// TwinCAT 3 PLC project Slider
// ProgramVersion: 3.1.4024.0
// libraries:
//   Tc2_MC2, * (Beckhoff Automation GmbH)
//   Tc2_Standard, * (Beckhoff Automation GmbH)
//   Tc2_System, * (Beckhoff Automation GmbH)
//   Tc3_Module, * (Beckhoff Automation GmbH)
// project tree:
//   DUTs/Cell/ ST_CELL.TcDUT, E_CMD_CELL.TcDUT
//   DUTs/CM/ E_CM_SERVO_CMD.TcDUT, ST_CM_SERVO.TcDUT, ST_CM_SERVO_CMD.TcDUT, ST_CM_SERVO_STS.TcDUT
//   DUTs/CM/Servo/ fbCmServo.TcPOU
//   DUTs/EM/ E_CMD.TcDUT, E_Function.TcDUT, E_Status.TcDUT, ST_CONFIG.TcDUT, ST_DATA.TcDUT, ST_EM.TcDUT, ST_MACHINE.TcDUT
//   DUTs/UN/ ST_UN.TcDUT
//   DUTs/UTIL/ E_DIRECTION.TcDUT, E_pos.TcDUT, STATUS_HMI.TcDUT
//   / GlobalTextList.TcGTLO, PlcTask.TcTTO, Visualization Manager.TcVMO (not stored)
//   GVLs/ Counters.TcGVL, GVL.TcGVL
//   POUs/ MAIN.TcPOU
//   POUs/Module/ fbEM.TcPOU, fbSliderEM.TcPOU, fbSliderWithGripperEM.TcPOU, fbXYMoverEM.TcPOU
//   POUs/Sim/ fbSignalSimPiotr.TcPOU, fbSignalSimSlider.TcPOU, fbSignalSimSliderWithGripper.TcPOU, fbSignalSimXYMover.TcPOU
//   POUs/UN/ fbTaskPatrykUN.TcPOU, fbTaskPiotrUN.TcPOU, fbUN.TcPOU
//   VISUs/ VisuPiotrUN.TcVIS
// real-time tasks:
//   TASK PlcTask: cycle T#10ms, priority 20, ADS port 350
// motion (NC):
//   TASK NC-Task 1 SAF: cycle T#2ms, priority 4, ADS port 501
//   TASK NC-Task 1 SVB: cycle T#10ms, priority 8, ADS port 511
//   AXIS Axis 1 (id 1)
//     OtherSettings: AllowMotionCmdToSlave=true
//     encoder EncType=1
//     drive DrvType=5
//       Analog: TorqueSetpointScale=10, ScaleFactorActTorque=0.1
//       TimeComp: TaskDelayCycles=1
//     controller CtrType=1
//       CtrPara: PriorControlFactor=1
//         Observer: BandWidth=20

CONFIGURATION Slider
    RESOURCE PLC ON TwinCAT3
        TASK PlcTask(INTERVAL := T#10ms, PRIORITY := 20);
        PROGRAM MAIN WITH PlcTask : MAIN;
    END_RESOURCE
END_CONFIGURATION

// ---- DUTs/Cell/ST_CELL.TcDUT
TYPE ST_CELL :
STRUCT
	Cmd : E_CMD_CELL;
	PlaceObject : ARRAY[1..5] OF BOOL; 
END_STRUCT
END_TYPE

// ---- DUTs/Cell/E_CMD_CELL.TcDUT
{attribute 'qualified_only'}
{attribute 'strict'}
TYPE E_CMD_CELL :
(
	STOP := 0,
	START,
	ABORT
);
END_TYPE

// ---- DUTs/CM/E_CM_SERVO_CMD.TcDUT
{attribute 'qualified_only'}
{attribute 'strict'}
TYPE E_CM_SERVO_CMD :
(
	idle := 0,
	reset,
	powerDisable,
	powerEnable,
	brakeDisable,
	brakeEnable,
	halt,
	moveVel,
	moveRel,
	moveAbs,
	moveMod,
	moveHome,
	jogP,
	jogN,
	jogStop
);
END_TYPE

// ---- DUTs/CM/ST_CM_SERVO.TcDUT
TYPE ST_CM_SERVO :
STRUCT
	cmd: ST_CM_SERVO_CMD;
	sts: ST_CM_SERVO_STS;
END_STRUCT
END_TYPE

// ---- DUTs/CM/ST_CM_SERVO_CMD.TcDUT
TYPE ST_CM_SERVO_CMD :
STRUCT
	cmd : E_CM_SERVO_CMD;
	start : BOOL;
END_STRUCT
END_TYPE

// ---- DUTs/CM/ST_CM_SERVO_STS.TcDUT
TYPE ST_CM_SERVO_STS :
STRUCT
	done: BOOL;
	outPos: BOOL;
	nearPos: BOOL;
	homed: BOOL;
	power: BOOL;
	error: BOOL;
	errorCode: UDINT;
	pos: REAL;
END_STRUCT
END_TYPE

// ---- DUTs/EM/E_CMD.TcDUT
// Enumerator containing em commands
{attribute 'qualified_only'}
{attribute 'strict'}
TYPE E_CMD :
(
	reset:=1,
	start,
	stop,
	hold,
	unhold,
	suspend,
	unsuspend,
	abort,
	clear,
	powerOn
);
END_TYPE

// ---- DUTs/EM/E_Function.TcDUT
// Enumerator containing general function of module
{attribute 'qualified_only'}
{attribute 'strict'}
{attribute 'to_string'}
TYPE E_Function :
(
	None,
	eSlider,
	eSliderWithGripper,
	eXYMover
);
END_TYPE

// ---- DUTs/EM/E_Status.TcDUT
// Enumerator contains packml state, unfortunatly named status
{attribute 'qualified_only'}
{attribute 'strict'}
TYPE E_Status :
(
	undefined:=0,
	clearing,
	stopped,
	starting,
	idle,
	suspended,
	execute,
	stopping,
	aborting,
	aborted,
	holding,
	held,
	unholding,
	suspending,
	unsuspending,
	resetting,
	completing,
	completed
);
END_TYPE

// ---- DUTs/EM/ST_CONFIG.TcDUT
// Structure config
{attribute 'qualified_only'}
{attribute 'strict'}
TYPE ST_CONFIG :
STRUCT
	Functionality : E_Function;
	Data : ST_DATA;
END_STRUCT
END_TYPE

// ---- DUTs/EM/ST_DATA.TcDUT
// Structure data contains inputs/outputs/axies
TYPE ST_DATA :
STRUCT
	I : REFERENCE TO ARRAY[1..10] OF BOOL;
	Q : REFERENCE TO ARRAY[1..10] OF BOOL;
	Axis : ARRAY[1..10] OF AXIS_REF;
	pick_pos :INT ; 					// Q CMD from where girpper picks
	drop_pos: INT ;						// Q CMD to where gripper moves for drop
	act_pos: INT;						// I actual position from of gripper
	give_pos: INT;						// writes value to servo_handle // simulator 
	takeObject : BOOL;
	objectSensor : BOOL;
END_STRUCT
END_TYPE

// ---- DUTs/EM/ST_EM.TcDUT
// Base structure em
TYPE ST_EM :
STRUCT
	Config : ST_CONFIG;
	Cmd : E_CMD;
	Status : E_Status;
	SequenceStep: INT;
	StatusHMI : STATUS_HMI;
END_STRUCT
END_TYPE

// ---- DUTs/EM/ST_MACHINE.TcDUT
// Utility structure to reference to fbEM
TYPE ST_MACHINE :
STRUCT
	fbEM : REFERENCE TO fbEM;
END_STRUCT
END_TYPE

// ---- DUTs/UN/ST_UN.TcDUT
// For now empty structure to build master for em-s
TYPE ST_UN :
STRUCT
	Cmd : E_CMD;
	Status : E_Status;
END_STRUCT
END_TYPE

// ---- DUTs/UTIL/E_DIRECTION.TcDUT
{attribute 'qualified_only'}
{attribute 'strict'}
TYPE E_DIRECTION :
(
	Left,
	Right,
	Up,
	Down,
	Downstream,
	Upstream
);
END_TYPE

// ---- DUTs/UTIL/E_pos.TcDUT
{attribute 'qualified_only'}
{attribute 'strict'}
TYPE E_pos :
(
	base := 0,
	one,
	two,
	three,
	four
	
);
END_TYPE

// ---- DUTs/UTIL/STATUS_HMI.TcDUT
TYPE STATUS_HMI :
STRUCT
	isMoving : BOOL;
	movingToPosition : INT;
	currentPosition : INT;
	movingDirection : E_DIRECTION;
	hasObject : BOOL;
	alarm : BOOL;
	alarmText : STRING;
	undefined : BOOL;
END_STRUCT
END_TYPE

// ---- GVLs/Counters.TcGVL
{attribute 'qualified_only'}
VAR_GLOBAL CONSTANT
	SliderEMNo : INT := 1;
	SliderWithGripperEMNo : INT := 1;
	XYMoverEMNo : INT := 2;
	
	packmlUnLast : INT := 1;
	packmlEmLast : INT := SliderEMNo + SliderWithGripperEMNo + XYMoverEMNo;
END_VAR

// ---- GVLs/GVL.TcGVL
// Global list with inputs/outputs to control and force variables
{attribute 'qualified_only'}
VAR_GLOBAL
	axis : AXIS_REF;
	aInput : ARRAY[1..10] OF ARRAY[1..10] OF BOOL;
	aOutput : ARRAY[1..10] OF ARRAY[1..10] OF BOOL;
	
	Input : ARRAY[1..10] OF BOOL;
	Output : ARRAY[1..10] OF BOOL;
END_VAR

// ---- POUs/MAIN.TcPOU
PROGRAM MAIN
VAR
	un : ST_UN;
	cell : ST_CELL;
	fbTaskPiotrUN : fbTaskPiotrUN;
	
	fb : fbSliderEM;
	em : ST_EM;
	
	START : BOOL;
	STOP : BOOL;
	ABORT : BOOL;
END_VAR

//cell.Cmd := E_CMD_CELL.START; 	// Selected as constant START to work in loop
//cell.PlaceObject := TRUE;		// Selected as constant placing object at input to work in loop

IF START THEN
	cell.Cmd := E_CMD_CELL.START;
	START := FALSE;
ELSIF STOP THEN
	cell.Cmd := E_CMD_CELL.STOP;
	STOP := FALSE;
ELSIF ABORT THEN
	cell.Cmd := E_CMD_CELL.ABORT;
	ABORT := FALSE;
END_IF

fbTaskPiotrUN(un := un, cell := cell, EnableSim := TRUE);

END_PROGRAM

// ---- POUs/UN/fbTaskPiotrUN.TcPOU
FUNCTION_BLOCK fbTaskPiotrUN EXTENDS fbUN
VAR
	// Arrays with 'em' universal structure and 'fbEM' containing ST_MACHINE structure which contains of references to fbEM function block
	em : ARRAY[1..Counters.packmlEmLast] OF ST_EM;
	fbEM : ARRAY[1..Counters.packmlEmLast] OF ST_MACHINE;
	
	// Array containing all instances fo fbSliderEM with its own iterator
	SliderEM : ARRAY[1..Counters.SliderEMNo] OF fbSliderEM;
	iSliderEM : DINT := 1;
	
	// Array containing all instances fo fbSliderWithGripperEM with its own iterator
	SliderWithGripperEM : ARRAY[1..Counters.SliderWithGripperEMNo] OF fbSliderWithGripperEM;
	iSliderWithGripperEM : DINT := 1;
	
	// Array containing all instances fo fbXYMoverEM with its own iterator
	XYMoverEM : ARRAY[1..Counters.XYMoverEMNo] OF fbXYMoverEM;
	iXYMoverEM : DINT := 1;
	
	fbSignalSimPiotr : fbSignalSimPiotr;
	
	i : DINT;
	j : DINT;
	State : INT := 0;
	StoppedState : INT := 0;
	declareIterator : DINT;
	moduleWorkIterator : DINT;
	initialConfig: BOOL := TRUE;
	svTime : TIME := T#15S;
	oTime : TIME := T#1S;
	supervisionTimer: TON;
	objectTimer: TON;
	objectWhichStopped : DINT := 0;
	takeObjectCounter : USINT;
	stoppedBy : STRING := '';
	stoppedByTemp : STRING;
	oneAlarm: BOOL;
END_VAR

// fbEM and em array number:
// 1 <- XYMovers
// 2 <- SliderWithGripper
// 3 <- XYMover
// 4 <- Slider
// 5 <- Slider

////////////////////////////////////////////////////////////////////////////////////////////////////////////////////////////
// All init configuration done here
IF initialConfig THEN
	initialConfig := FALSE;
	// Specifing module type of each module in array
	em[1].Config.Functionality := E_Function.eXYMover;
	em[2].Config.Functionality := E_Function.eSliderWithGripper;
	em[3].Config.Functionality := E_Function.eXYMover;
	em[4].Config.Functionality := E_Function.eSlider;
	em[5].Config.Functionality := E_Function.eSlider;

	// FOR loop to specify config for each module
	FOR declareIterator := 1 TO Counters.packmlEmLast DO
		em[declareIterator].Config.Data.I REF= GVL.aInput[declareIterator];
		em[declareIterator].Config.Data.Q REF= GVL.aOutput[declareIterator];

		CASE em[declareIterator].Config.Functionality OF
			E_Function.eSlider:
				fbEM[declareIterator].fbEM REF= SliderEM[iSliderEM];
				iSliderEM := iSliderEM + 1;
			E_Function.eSliderWithGripper:
				fbEM[declareIterator].fbEM REF= SliderWithGripperEM[iSliderWithGripperEM];
				iSliderWithGripperEM := iSliderWithGripperEM + 1;
			E_Function.eXYMover:
				fbEM[declareIterator].fbEM REF= XYMoverEM[iXYMoverEM];
				iXYMoverEM := iXYMoverEM + 1;
		END_CASE
	END_FOR
	
	em[2].Config.Data.pick_pos := 3;
	em[2].Config.Data.drop_pos := 2;
	
	supervisionTimer.PT := svTime;
	objectTimer.PT := oTime;
END_IF

////////////////////////////////////////////////////////////////////////////////////////////////////////////////////////////
// Modules work loop (idk yet if is better to have it at the beggining or bottom of UN)
FOR moduleWorkIterator := 1 TO Counters.packmlEmLast DO
	fbEM[moduleWorkIterator].fbEM(em := em[moduleWorkIterator], un := un, EnableSim := EnableSim, CmdSim := FALSE);
END_FOR

////////////////////////////////////////////////////////////////////////////////////////////////////////////////////////////

fbSignalSimPiotr(em := em, State := State, EnableSim := EnableSim);

IF supervisionTimer.Q THEN
	stoppedBy := 'Supervision';
	supervisionTimer(IN := FALSE);
	cell.Cmd := E_CMD_CELL.STOP;
END_IF

FOR j := 1 TO Counters.packmlEmLast DO
	IF NOT em[j].Config.Data.takeObject AND em[j].Config.Data.objectSensor THEN
		objectTimer(IN := TRUE);
		objectWhichStopped := j;
	ELSIF objectWhichStopped = j
	AND ((em[j].Config.Data.takeObject AND em[j].Config.Data.objectSensor)
	OR (NOT em[j].Config.Data.takeObject AND NOT em[j].Config.Data.objectSensor)) THEN
		objectWhichStopped := 0;
		objectTimer(IN := FALSE);
		oneAlarm := FALSE;
	END_IF
END_FOR

IF objectTimer.Q THEN
	cell.Cmd := E_CMD_CELL.STOP;
	IF NOT oneAlarm THEN
		stoppedBy := CONCAT('Object at em: ', DINT_TO_STRING(ObjectWhichStopped));
		oneAlarm := TRUE;
	END_IF
END_IF

IF cell.Cmd = E_CMD_CELL.STOP AND State < 2000 THEN
	StoppedState := State;
	State := 2000;
END_IF

IF cell.Cmd = E_CMD_CELL.ABORT AND State < 1000 THEN
	stoppedBy := 'ABORT Button';
	StoppedState := 0;
	State := 1000;
END_IF

CASE State OF
	0:	un.Status := E_Status.undefined;
		em[2].Config.Data.pick_pos := 3;
		em[2].Config.Data.drop_pos := 2;
		State := 5;
	
	5:	// Waiting for every EM to become idle state
		FOR i := 1 TO Counters.packmlEmLast DO
			IF NOT (em[i].Status = E_Status.idle) THEN
				un.Cmd := E_CMD.reset;
				RETURN;
			END_IF
		END_FOR
		un.Status := E_Status.idle;
		State := 10;
	
	10:	IF cell.Cmd = E_CMD_CELL.START THEN
			stoppedBy := '';
			un.Cmd := E_CMD.start;
			un.Status := E_Status.starting;
			State := 20;
		END_IF
	
	20:	// Waiting for every EM to be in execute or starting state
		FOR i := 1 TO Counters.packmlEmLast DO
			IF NOT (em[i].Status = E_Status.execute OR em[i].Status = E_Status.starting) THEN
				RETURN;
			END_IF
		END_FOR
		State := 30;
		
	30:	// Start of my specific task (all modules stays in execute)
		// input -> XY1 -> SWG -> XY2 -> S1 -> SWG -> S2 -> output
		IF (em[1].SequenceStep = 20		// XY1
		AND cell.PlaceObject)			// Object input signal
		THEN
			cell.PlaceObject := FALSE;
			em[1].Config.Data.takeObject := TRUE;
			State := 40;
		END_IF
		
		IF StoppedState <> 0 AND StoppedState < 1000 THEN
			State := StoppedState;
			StoppedState := 0;
		END_IF
		
	40:	// XY1 -> SWG -> XY2 -> S1 -> SWG -> S2 -> output
		supervisionTimer(IN := TRUE);
		
		IF em[1].SequenceStep = 60		// XY1
		AND em[2].SequenceStep = 40		// SWG
		THEN
			em[1].Config.Data.takeObject := FALSE;
			em[2].Config.Data.takeObject := TRUE;
			
			State := 50;
			supervisionTimer(IN := FALSE);
		END_IF
		
	50: // SWG -> XY2 -> S1 -> SWG -> S2 -> output
		supervisionTimer(IN := TRUE);
		
		IF em[2].SequenceStep = 43		// SWG
		AND em[3].SequenceStep = 20		// XY2
		THEN
			em[2].Config.Data.takeObject := FALSE;
			em[3].Config.Data.takeObject := TRUE;
			
			em[2].Config.Data.pick_pos := 4;
			State := 60;
			supervisionTimer(IN := FALSE);
		END_IF
		
	60: // XY2 -> S1 -> SWG -> S2 -> output
		supervisionTimer(IN := TRUE);
		
		IF em[3].SequenceStep = 60		// XY2
		AND em[4].SequenceStep = 50		// S1
		THEN
			em[3].Config.Data.takeObject := FALSE;
			em[4].Config.Data.takeObject := TRUE;
			
			em[2].Config.Data.drop_pos := 1;
			State := 70;
			supervisionTimer(IN := FALSE);
		END_IF
		
	70:	// S1 -> SWG -> S2 -> output
		supervisionTimer(IN := TRUE);
		
		IF em[2].SequenceStep = 40		// SWG
		AND em[4].SequenceStep = 70		// S1
		THEN
			em[4].Config.Data.takeObject := FALSE;
			em[2].Config.Data.takeObject := TRUE;
			
			State := 80;
			supervisionTimer(IN := FALSE);
		END_IF
		
	80:	// SWG -> S2 -> output
		supervisionTimer(IN := TRUE);
		
		IF em[2].SequenceStep = 43		// SWG
		AND em[5].SequenceStep = 50		// S2
		THEN
			em[2].Config.Data.takeObject := FALSE;
			em[5].Config.Data.takeObject := TRUE;
			
			em[2].Config.Data.pick_pos := 3;
			State := 90;
			supervisionTimer(IN := FALSE);
		END_IF
		
	90:	// S2 -> output
		supervisionTimer(IN := TRUE);
		IF em[5].SequenceStep = 70 THEN
			em[2].Config.Data.drop_pos := 2;
			State := 100;
			supervisionTimer(IN := FALSE);
		END_IF
		
	100: // output
		IF NOT em[5].Config.Data.objectSensor THEN
			em[5].Config.Data.takeObject := FALSE;
			State := 30;
		END_IF
		
	1000:
		un.Cmd := E_CMD.abort;
		un.Status := E_Status.aborting;
		FOR i := 1 TO Counters.packmlEmLast DO
			IF NOT (em[i].Status = E_Status.aborted) THEN
				RETURN;
			END_IF
		END_FOR
		State := 1010;
	
	1010:
		IF cell.Cmd = E_CMD_CELL.START THEN
			un.Cmd := E_CMD.clear;
			State := 2000;
		END_IF

	2000:
		un.Cmd := E_CMD.stop;
		un.Status := E_Status.stopping;
		supervisionTimer(IN := FALSE);
		objectTimer(IN := FALSE);
		FOR i := 1 TO Counters.packmlEmLast DO
			IF em[i].Status <> E_Status.stopped THEN
				RETURN;
			END_IF
		END_FOR
		un.Status := E_Status.stopped;
		State := 2010;
	
	2010:
		IF cell.Cmd = E_CMD_CELL.START THEN
			State := 5;
		END_IF	
END_CASE

// Do not write anything here, it will not execute everytime due to RETURN command used in case

END_FUNCTION_BLOCK

// ---- POUs/UN/fbUN.TcPOU
FUNCTION_BLOCK fbUN
VAR_IN_OUT
	un : ST_UN;
	cell : ST_CELL;
END_VAR
VAR_INPUT
	EnableSim : BOOL;
END_VAR

END_FUNCTION_BLOCK

// ---- POUs/Module/fbEM.TcPOU
FUNCTION_BLOCK fbEM
VAR_IN_OUT
	em : ST_EM;
	un : ST_UN;
END_VAR

VAR_INPUT
	EnableSim : BOOL;
	CmdSim : BOOL := TRUE;
END_VAR

VAR
	emCmdOld: E_CMD;
END_VAR

// Empty for now universal basic em class, every module needs to extends this to ensure compatibility

ACTION GetUnCmd:
IF emCmdOld <> un.Cmd THEN
	emCmdOld := un.Cmd;
	em.Cmd := un.Cmd;
END_IF
END_ACTION

END_FUNCTION_BLOCK

// ---- POUs/Module/fbSliderEM.TcPOU
FUNCTION_BLOCK fbSliderEM EXTENDS fbEM
VAR_INPUT
	UnknownStartPosition : BOOL := FALSE;
	StartOnOtherSide : BOOL := FALSE;
END_VAR

VAR
	bSliderSide : BOOL;
	XYMoverActualStep: INT;
	fbSignalSim : fbSignalSimSlider;
	timer : TON;
	timerPT : TIME := T#2S;
END_VAR

VAR RETAIN
	State : INT := 0;
END_VAR

(*
	Input/Output mapping
	I[1] <- Siłownik pozycja 1 (wsunięty) 
	I[2] <- Siłownik pozycja 2 (wysunięty)
	I[3] <- Czujnik obecności obiektu (na pozycji 1 (wsunięty)) 
	Q[1] <- Wysuń siłownik (do pozycji 2)
	Q[2] <- Wsuń siłownik (do pozycji 1)
*)

GetUnCmd();
fbSignalSim(
	em := em,
	EnableSim := EnableSim,
	UnknownStartPosition := UnknownStartPosition,
	StartOnOtherSide := StartOnOtherSide,
	CmdSim := CmdSim
);
timer(PT := timerPT);

IF em.Config.Functionality = E_Function.eSlider THEN
	IF State >= 15 AND em.Cmd = E_CMD.abort THEN
		State := 5;
	END_IF
	
	IF State >= 35 AND em.Cmd = E_CMD.stop THEN
		State := 15;
	END_IF

	CASE State OF
		0:	em.StatusHMI.isMoving := FALSE;
			em.StatusHMI.undefined := TRUE;
			IF em.Config.Data.I[1] OR em.Config.Data.I[2] THEN
				State := 1;
				em.StatusHMI.undefined := FALSE;
			ELSE
				em.Status := E_Status.undefined;
				State := 20;
			END_IF
			
		1:	IF em.Config.Data.I[2] THEN
				bSliderSide := TRUE;
				em.StatusHMI.currentPosition := 2;
			ELSE
				em.StatusHMI.currentPosition := 1;
			END_IF
			State := 40;
		
		5:	em.Status := E_Status.aborting;
			em.Config.Data.Q[1] := FALSE;
			em.Config.Data.Q[2] := FALSE;
			em.StatusHMI.isMoving := FALSE;
			em.StatusHMI.undefined := TRUE;
			State := 7;
			
		7:	em.Status := E_Status.aborted;
			State := 10;
			
		10:	IF em.Cmd = E_CMD.clear THEN
				em.Status := E_Status.clearing;
				em.StatusHMI.undefined := FALSE;
				State := 20;
			END_IF
			
		15: em.Status := E_Status.stopping;
			em.Config.Data.Q[1] := FALSE;
			em.Config.Data.Q[2] := FALSE;
			em.StatusHMI.isMoving := FALSE;
			em.StatusHMI.undefined := FALSE;
			State := 20;
			
		20:	em.Status := E_Status.stopped;
			State := 30;
			
		30:	IF em.Cmd = E_CMD.reset THEN
				em.Status := E_Status.resetting;
				em.Config.Data.Q[1] := FALSE;
				em.Config.Data.Q[2] := TRUE;
				em.StatusHMI.isMoving := TRUE;
				em.StatusHMI.movingDirection := E_DIRECTION.Upstream;
				em.StatusHMI.movingToPosition := 1;
				State := 35;
			END_IF
			
		35:	IF em.Config.Data.I[1] THEN
				em.StatusHMI.isMoving := FALSE;
				em.Config.Data.Q[2] := FALSE;
				bSliderSide := FALSE;
				State := 40;
			END_IF
			
		40:	em.Status := E_Status.idle;
			IF em.Cmd = E_CMD.start THEN
				State := 45;
			END_IF
			
		45:	em.Status := E_Status.Starting;
			State := 50;
			
			// Execute direction
		50:	em.Status := E_Status.execute;
			IF bSliderSide AND NOT em.Config.Data.I[3] THEN
				timer(IN := TRUE);
				State := 52;
			ELSIF em.Config.Data.I[3] THEN
				timer(IN := TRUE);
				State := 55;
			END_IF
			
		52: IF timer.Q THEN
				em.StatusHMI.movingDirection := E_DIRECTION.Upstream;
				em.StatusHMI.movingToPosition := 1;
				em.StatusHMI.undefined := FALSE;
				timer(IN := FALSE);
				em.Config.Data.Q[2] := TRUE;
				State := 60;
			END_IF	
			
		55: IF timer.Q THEN
				em.StatusHMI.movingDirection := E_DIRECTION.Downstream;
				em.StatusHMI.movingToPosition := 2;
				em.StatusHMI.undefined := FALSE;
				timer(IN := FALSE);
				em.Config.Data.Q[1] := TRUE;
				State := 60;
			END_IF	
			
			// Main execute
		60:	IF em.Cmd = E_CMD.hold THEN
				em.StatusHMI.undefined := TRUE;
				em.Status := E_Status.holding;
				State := 200;
			ELSIF em.Cmd = E_CMD.suspend THEN
				em.StatusHMI.undefined := TRUE;
				em.Status := E_Status.suspending;
				State := 300;
			END_IF
			
			IF em.Config.Data.Q[2] AND em.Config.Data.I[1] THEN
				em.Config.Data.Q[2] := FALSE;
				bSliderSide := FALSE;
				State := 50;
			END_IF
			
			IF em.Config.Data.Q[1] AND em.Config.Data.I[2] THEN
				bSliderSide := TRUE;
				State := 70;
			END_IF
			
		70:	IF NOT em.Config.Data.I[3] THEN
				em.Config.Data.Q[1] := FALSE;
				State := 50;
			END_IF
			
		200:em.Status := E_Status.held;
			em.Config.Data.Q[1] := FALSE;
			em.Config.Data.Q[2] := FALSE;
			em.StatusHMI.undefined := TRUE;
			IF em.Cmd = E_CMD.unhold THEN
				em.Status := E_Status.unholding;
				State := 50;
			END_IF
			
		300:em.Status := E_Status.suspended;
			em.Config.Data.Q[1] := FALSE;
			em.Config.Data.Q[2] := FALSE;
			em.StatusHMI.undefined := TRUE;
			IF em.Cmd = E_CMD.unsuspend THEN
				em.Status := E_Status.unsuspending;
				State := 50;
			END_IF
	END_CASE
END_IF

em.SequenceStep := State;
em.Config.Data.objectSensor REF= em.Config.Data.I[3];

IF em.Config.Data.Q[1] XOR em.Config.Data.Q[2] THEN
	em.StatusHMI.isMoving := TRUE;
ELSIF em.Config.Data.Q[1] AND em.Config.Data.Q[2] THEN
	em.StatusHmi.isMoving := FALSE;
	em.StatusHMI.undefined := TRUE;
	em.StatusHMI.alarm := TRUE;
	em.StatusHMI.alarmText := 'Both actuators are operating';
ELSE
	em.StatusHmi.isMoving := FALSE;
	em.StatusHMI.undefined := FALSE;
	em.StatusHMI.alarm := FALSE;
	em.StatusHMI.alarmText := '';
END_IF

IF em.Config.Data.I[3] THEN
	em.StatusHMI.hasObject := TRUE;
ELSE
	em.StatusHMI.hasObject := FALSE;
END_IF

IF em.Config.Data.I[1] THEN
	em.StatusHMI.currentPosition := 1;
ELSIF em.Config.Data.I[2] THEN
	em.StatusHMI.currentPosition := 2;
ELSE
	em.StatusHMI.currentPosition := 0;
END_IF

END_FUNCTION_BLOCK

// ---- POUs/Sim/fbSignalSimSlider.TcPOU
FUNCTION_BLOCK fbSignalSimSlider
VAR_IN_OUT
	em : ST_EM;
END_VAR
VAR_INPUT
	EnableSim : BOOL;
	UnknownStartPosition : BOOL := FALSE;
	StartOnOtherSide : BOOL := FALSE;
	CmdSim : BOOL := true;
END_VAR
VAR
	InitialConfig : BOOL := TRUE;
	timers : ARRAY[1..10] OF TON;
	duration : TIME := T#5S;
	elapsed : TIME;
	OtherSide : BOOL := FALSE;
END_VAR

IF EnableSim THEN
	IF InitialConfig THEN
		InitialConfig := FALSE;
		IF NOT UnknownStartPosition THEN
			IF StartOnOtherSide THEN
				em.Config.Data.I[2] := TRUE;
				OtherSide := TRUE;
			ELSE
				em.Config.Data.I[1] := TRUE;
			END_IF
		ELSE
			em.Config.Data.I[1] := FALSE;
			em.Config.Data.I[2] := FALSE;
		END_IF
		
		timers[1].PT := timers[2].PT := timers[3].PT := timers[10].PT := duration;
		timers[4].PT := timers[5].PT := timers[6].PT := timers[7].PT := timers[8].PT := timers[9].PT := duration / 3;
	END_IF
	
	CASE em.SequenceStep OF
		10:	IF CmdSim THEN
				timers[5](in := TRUE);
			
				IF timers[5].Q THEN
					timers[5](in := FALSE);
					em.Cmd := E_CMD.clear;
				END_IF
			END_IF
	
		30:	IF CmdSim THEN
				timers[6](in := TRUE);
			
				IF timers[6].Q THEN
					timers[6](in := FALSE);
					em.Cmd := E_CMD.reset;	
				END_IF
			END_IF

		35:	timers[10](in := TRUE);
		
			IF timers[10].Q THEN
				timers[10](in := FALSE);
				em.Config.Data.I[1] := TRUE;
			END_IF
	
		40: IF CmdSim THEN
				timers[4](in := TRUE);
			
				IF timers[4].Q THEN
					timers[4](in := FALSE);
					em.Cmd := E_CMD.start;
				END_IF
			END_IF

		50:	IF CmdSim THEN
				IF NOT OtherSide AND em.Config.Data.I[1] THEN
					timers[1](in := TRUE); 
				END_IF
				
				IF timers[1].Q THEN
					timers[1](in := FALSE);
					em.Config.Data.I[3] := TRUE;
				END_IF
			END_IF
			
		60:	IF NOT OtherSide AND em.Config.Data.I[1] THEN
				timers[2](in := NOT timers[2].Q);
				em.Config.Data.I[1] := FALSE;
				em.Config.Data.I[2] := FALSE;
			ELSE
				timers[3](in := NOT timers[3].Q);
				em.Config.Data.I[1] := FALSE;
				em.Config.Data.I[2] := FALSE;
			END_IF
			
			IF timers[2].Q THEN
				timers[2](in := FALSE);
				em.Config.Data.I[2] := TRUE;
			END_IF
			
			IF timers[3].Q THEN
				timers[3](in := FALSE);
				em.Config.Data.I[1] := TRUE;
			END_IF
			
		70:	IF CmdSim THEN
				timers[1](in := TRUE);
				
				IF timers[1].Q THEN
					timers[1](in := FALSE);
					em.Config.Data.I[3] := FALSE;
				END_IF
			END_IF
			
		200:IF CmdSim THEN
				timers[8](in := TRUE);
			
				IF timers[8].Q THEN
					timers[8](in := FALSE);
					em.Cmd := E_CMD.unhold;	
				END_IF
			END_IF
		
		300:IF CmdSim THEN
				timers[9](in := TRUE);
			
				IF timers[9].Q THEN
					timers[9](in := FALSE);
					em.Cmd := E_CMD.unsuspend;	
				END_IF
			END_IF
	END_CASE

	OtherSide := FALSE;
END_IF

END_FUNCTION_BLOCK

// ---- POUs/Module/fbSliderWithGripperEM.TcPOU
FUNCTION_BLOCK fbSliderWithGripperEM EXTENDS fbEM
VAR
	i : INT;
	state : INT;
	initial: BOOL := TRUE;
	servo_GO: BOOL;
	
	fbSignalSim: fbSignalSimSliderWithGripper;
END_VAR
VAR_INPUT
	
END_VAR
VAR_OUTPUT
	
END_VAR

(*
THIS fb use IOs listed below
DATA.I[1] -> true when gripper closed
DATA.I[2] -> true when gripper opened
DATA.I[3] -> part present
DATA.Q[1] -> 1 CLOSE / 0 OPEN gripper
DATA.Q[3] -> SERVO_GO
DATA.pick_pos -> desired pick position
DATA.drop_pos -> desired drop position
DATA.act_pos -> actual postition ( resolved in SIM or SERVO_HANDLER)
DATA.give_pos -> moves desired position into SIM or SERVO_HANDLER)
*)

GetUnCmd();
fbSignalSim(
	em := em,
	EnableSim := EnableSim,
	CmdSim := CmdSim
);

IF initial THEN // AFTER START OF PLC ENTER Undefined state
	state:=0;
	//em.CMD := E_CMD.powerOn; //// MAKES SENSE? <- no it doesnt because you change input 
	initial:= FALSE;
	//	 em.Config.Data.pick_pos:=10; 
	//	 em.Config.Data.pick_pos:=200;
	
END_IF

IF em.CMD = E_CMD.abort THEN
	state:=65;
END_IF

IF em.CMD = E_CMD.stop THEN
	state:=70;
END_IF

CASE state OF
	
	0:		//RESETTING
		em.Status := E_Status.resetting;	
		
		
		IF  em.Config.Data.pick_pos = em.Config.Data.act_pos THEN   // ACTUAL POS READ FROM SERVO HANDLER / FOR NOW FROM SIGNAL SIM
				
				servo_GO:=FALSE;
				state :=30; // IF gripper at PICK_pos go to idle
		END_IF
		IF em.CMD = E_CMD.reset THEN 		
				em.Config.Data.give_pos:=em.Config.Data.pick_pos;
				servo_GO:=TRUE;
				
				//// IF gripper pos unknown move to PICK
				//SERVO_HANDLER HAS TO KNOW THE CASE STEP TO DECIDE WHERE TO MOVE 			 
				//HERE SIGNAL SIM HANDLE THIS		
		END_IF
		

	
	30:		//IDLE
		em.Status := E_Status.idle;
		IF em.CMD = E_CMD.start THEN 
			state :=40;
		END_IF
		

	40:		//EXECUTE.1
		em.Status := E_Status.execute;
				
		//Close gripper when part present
		IF em.Config.Data.I[3]  THEN 
			em.Config.Data.Q[1]:= TRUE; //CLOSE GRIPPER
		END_IF
		
		//When Gripper closed --> state 41
		IF em.Config.Data.I[1] = TRUE AND em.Config.Data.I[2]=FALSE THEN
			state:=41;
		END_IF

	41:		//EXECUTE.2 ORDER TO MOVE TO CHOOSEN POSITION
		em.Status := E_Status.execute;
		em.Config.Data.give_pos := em.Config.Data.drop_pos;
		servo_GO:=TRUE; 							
		IF em.Config.Data.act_pos = em.Config.Data.drop_pos THEN
		servo_GO:=FALSE;
		state:=42;										
		END_IF


	42:		//EXECUTE.3 OPEN GRIPPER
	
		em.Status := E_Status.execute;
		em.Config.Data.Q[1]:=FALSE; //OPEN GRIPPER
		IF em.Config.Data.I[1] = FALSE AND em.Config.Data.I[2]=TRUE THEN
			state:=43;
		END_IF
		
			
	43:		//EXECUTE.4 MOVING PICK_POS WITHOUT PART

		em.Status := E_Status.execute;
		IF NOT em.Config.Data.I[3]  
			AND em.Config.Data.act_pos =em.Config.Data.drop_pos THEN//when part gone
			em.Config.Data.give_pos:=em.Config.Data.pick_pos;
			servo_GO:=TRUE;//GO 
			//SERVO_HANDLER HAS TO KNOW THE CASE STEP TO DECIDE WHERE TO MOVE 			 
			//HERE SIGNAL SIM HANDLE THIS	
		END_IF
		
		IF em.Config.Data.act_pos = em.Config.Data.pick_pos THEN
			servo_GO:=FALSE;
			state:=40;
			//em.Config.Data.pick_pos:= -1;
			//em.Config.Data.drop_pos:= -1;
		END_IF
	
	
	65:		//ABORTED

		em.Status := E_Status.aborted;	
		servo_GO:=FALSE;
		IF em.CMD = E_CMD.clear THEN
			state := 70;
		END_IF;


	70: //STOPPED

		em.Status := E_Status.stopped;	
		servo_GO:=FALSE;
		IF em.CMD = E_CMD.reset THEN
			state:=0;
		END_IF

	
END_CASE



em.SequenceStep:=state;       //pass sequence step outside to SimSignal

em.Config.Data.Q[3]:=servo_GO;//Q[3] alias
em.Config.Data.objectSensor REF= em.Config.Data.I[3];




(*  SERVO HANDLER LOGIC
	IF SERVO_GO AND STATE = 0 THEN MOVE_TO_PICK_POS
	IF SERVO_GO AND STATE = 41 THEN MOVE_TO_DROP_POS
	IF SERVO_GO AND STATE = 44 THEN MOVE_TO_PICK_POS  *)

(*BEST MOMENT TO WRITE DESIRED pick_pos or drop_pos is STATE 30 or 40*)

END_FUNCTION_BLOCK

// ---- POUs/Sim/fbSignalSimSliderWithGripper.TcPOU
FUNCTION_BLOCK fbSignalSimSliderWithGripper
VAR_IN_OUT
	em : ST_EM; 
END_VAR
VAR_INPUT
	EnableSim : BOOL;
	CmdSim : BOOL := true;
END_VAR
VAR
	 
	i : int; 
	delay: ARRAY [1..10] OF TON;
END_VAR

delay[1](PT:=T#2S); delay[1].ET;//Open GRIPPER Movement Sim
delay[2](PT:=T#2S); delay[2].ET;//Close GRIPPER Movement SIm
delay[3](PT:=T#5S); delay[3].ET;// Moving  PICK_POS //DROP_POS
delay[4](PT:=T#4S); delay[4].ET;//CMD.Clear simulation
delay[5](PT:=T#4S); delay[5].ET;
delay[6](PT:=T#4S); delay[6].ET;
delay[7](PT:=T#4S); delay[7].ET;//OpenGRipp State 0
delay[9](PT:=T#2S); delay[9].ET;//CMD.clear
delay[10](PT:=T#2S);delay[10].ET;//CMD.reset

IF EnableSim THEN
		
	IF em.Cmd = E_CMD.abort THEN
		delay[9](IN:=TRUE);
	END_IF
	
	IF em.Cmd = E_CMD.stop THEN
		delay[10](IN:=TRUE);
	END_IF
	
	
	
	CASE em.SequenceStep OF
		
		0:		//Undefined state
				
			
				//Simulate CMD.clear button
			IF CmdSim THEN	
				IF delay[4].Q THEN
					delay[4](IN:=FALSE);
					em.Cmd:=E_CMD.reset;
				END_IF
				delay[4](IN:=TRUE);
			END_IF
				
				//Simulate movement to PICK_POS 
			IF em.Config.Data.Q[3]=TRUE THEN
				delay[3](IN:=TRUE);
			END_IF
			
			IF delay[3].Q THEN
					delay[3](IN:=FALSE);
					
					em.Config.Data.act_pos:=em.Config.Data.give_pos;	// Gripper position clear
					
			END_IF
	
			
			
			
		
		
		30:		//IDLE
				
				//WAIT FOR CMD
			IF CmdSim THEN				
				IF delay[6].Q THEN
					delay[6](IN:=FALSE);
					em.Cmd:=E_Cmd.start;
				END_IF
				delay[6](IN:=TRUE);
			END_IF
			
		40:		//EXECUTE.1
				
				//Simulate closing gripper
			IF em.Config.Data.Q[1]= TRUE THEN
				delay[2](IN:=TRUE);
			END_IF
			
			
			
			IF delay[2].Q THEN
				em.Config.Data.I[1]:= TRUE;
				em.Config.Data.I[2]:=FALSE;
				delay[2](IN:=FALSE);
			END_IF
		
	
		41:		//EXECUTE.2
				
			IF em.Config.Data.Q[3]=TRUE AND em.Config.Data.act_pos =em.Config.Data.pick_pos THEN  //servoGO		
				delay[3](IN:=TRUE);	
				em.Config.Data.act_pos:=666; //LEAVING HOME
			END_IF
				
			IF delay[3].Q THEN
				delay[3].IN:=FALSE;
				em.Config.Data.act_pos:= em.Config.Data.give_pos;		
			END_IF
		
		
		42:		//EXECUTE.3 OPEN GRIPPER
		
				//Simulate opening gripper
			IF em.Config.Data.Q[1]= FALSE  THEN
			delay[1](IN:=TRUE);
			
			END_IF
	 
			IF delay[1].Q THEN
				em.Config.Data.I[1]:= FALSE;
				em.Config.Data.I[2]:=TRUE;
				delay[1](IN:=FALSE);
			END_IF
		43:		//EXECUTE.4 MOVING PICK_pOS 
		
			IF em.Config.Data.Q[3]=TRUE AND
			em.Config.Data.act_pos =em.Config.Data.drop_pos THEN
				delay[3](IN:=TRUE);	
				em.Config.Data.act_pos:=666;
			END_IF
				
			IF delay[3].Q THEN
			delay[3].IN:=FALSE;
			em.Config.Data.act_pos:=em.Config.Data.give_pos; // arrived at pick_pos
			END_IF;
				
		65:		//ABORTED
			IF CmdSim THEN
				IF delay[9].Q THEN
				delay[9].IN:=FALSE;
				em.Cmd:=E_Cmd.clear;
				delay[10].IN:=TRUE;
				END_IF
			END_IF
		
		
		70:		//STOPPED
			IF CmdSim THEN
				IF delay[10].Q THEN
				delay[10].IN:=FALSE;
				em.Cmd:=E_Cmd.reset;
				END_IF
			END_IF
	END_CASE
	
END_IF

END_FUNCTION_BLOCK

// ---- POUs/Module/fbXYMoverEM.TcPOU
FUNCTION_BLOCK fbXYMoverEM EXTENDS fbEM
VAR_IN_OUT
END_VAR
VAR
	F_Reset : BOOL := TRUE;
	fbSignalSim: fbSignalSimXYMover;
END_VAR
VAR RETAIN
	XYMoverActualStep : INT;
END_VAR

GetUnCmd();
fbSignalSim(
	em := em,
	EnableSim := EnableSim,
	CmdSim := CmdSim
);

IF em.Config.Functionality = E_Function.eXYMover THEN
            IF XYMoverActualStep <> 2 AND XYMoverActualStep <> 3 AND XYMoverActualStep <> 4 AND em.Cmd = E_Cmd.STOP THEN
                   XYMoverActualStep := 1;
            END_IF
            IF XYMoverActualStep <> 6 AND XYMoverActualStep <> 7 AND XYMoverActualStep <> 2 AND XYMoverActualStep <> 3 AND XYMoverActualStep <> 4 AND em.Cmd = E_Cmd.ABORT THEN
                   XYMoverActualStep := 5;
           	END_IF


CASE XYMoverActualStep OF
	
	0: 		IF em.Config.Data.I[3] AND em.Config.Data.I[1] THEN
                  em.Status := E_Status.IDLE;
                  XYMoverActualStep := 10;
            ELSE 
                  em.Status := E_Status.UNDEFINED;
                  XYMoverActualStep := 2;
            END_IF
            
	1:      em.Status := E_Status.stopping;
            em.Config.Data.Q[1] := FALSE;
            em.Config.Data.Q[2] := FALSE;
            em.Config.Data.Q[3] := FALSE;
            em.Config.Data.Q[4] := FALSE;
            XYMoverActualStep := 2;
                        
	2:		em.Status := E_Status.stopped; 
            XYMoverActualStep := 3;
            
	3:  	IF em.Cmd = E_CMD.reset THEN
                 em.Status := E_Status.resetting;
                 em.Config.Data.Q[1] := TRUE;
                 em.Config.Data.Q[3] := TRUE;
				 em.Config.Data.Q[2] := FALSE;
				 em.Config.Data.Q[4] := FALSE;
                 XYMoverActualStep := 4;
            END_IF
                        
	4:      IF em.Config.Data.I[3] AND em.Config.Data.I[1] THEN
                 XYMoverActualStep := 0;
            END_IF
                           
	5:      em.Status := E_Status.aborting;
            em.Config.Data.Q[1] := FALSE;
            em.Config.Data.Q[2] := FALSE;
            em.Config.Data.Q[3] := FALSE;
            em.Config.Data.Q[4] := FALSE;
            XYMoverActualStep := 6;
			
	6:		em.Status := E_Status.aborted; 
            XYMoverActualStep := 7;
                        
	7:      IF em.Cmd = E_CMD.clear THEN
                em.Status := E_Status.clearing;
                XYMoverActualStep := 2;
            END_IF
                                                                                              
	10:		IF em.Cmd = E_Cmd.START THEN
                em.Status := E_Status.STARTING;
                XYMoverActualStep := 20;
            END_IF

	20:		em.Status := E_Status.EXECUTE;
			IF em.Config.Data.I[5] = TRUE THEN
                XYMoverActualStep := 30; 
            END_IF

	30:		em.Config.Data.Q[1] := FALSE;
            em.Config.Data.Q[2] := TRUE;
			IF em.Config.Data.I[2] = TRUE AND em.Config.Data.I[1] = FALSE THEN
           		XYMoverActualStep := 40;
			END_IF
            
	40:  
			em.Config.Data.Q[3] := FALSE;
			em.Config.Data.Q[4] := TRUE;
			IF em.Config.Data.I[4] = TRUE AND em.Config.Data.I[3] = FALSE THEN
				XYMoverActualStep := 50;
			END_IF
                        
	50:
            IF em.Config.Data.I[4] = TRUE THEN
                XYMoverActualStep := 60; 
            END_IF 
            
	60: 	IF em.Config.Data.I[5] = FALSE THEN
            	XYMoverActualStep := 70; 
            END_IF 
            
	70: 	em.Config.Data.Q[2] := FALSE;
			em.Config.Data.Q[4] := FALSE;
			em.Config.Data.Q[3] := TRUE;
            em.Config.Data.Q[1] := TRUE;
			IF em.Config.Data.I[1] = TRUE AND em.Config.Data.I[2] = FALSE AND em.Config.Data.I[3] = TRUE AND em.Config.Data.I[4] = FALSE THEN
				XYMoverActualStep := 20;
			END_IF
                        
END_CASE
END_IF

em.SequenceStep := XYMoverActualStep;
em.Config.Data.objectSensor REF= em.Config.Data.I[5];

END_FUNCTION_BLOCK

// ---- POUs/Sim/fbSignalSimXYMover.TcPOU
FUNCTION_BLOCK fbSignalSimXYMover
VAR_IN_OUT
	em : ST_EM;
END_VAR
VAR_INPUT
	EnableSim : BOOL;
	CmdSim : BOOL := true;
END_VAR
VAR
	TimerSim : Array[1..12] OF TON;
	Elapsed : TIME;
END_VAR

IF EnableSim THEN
	CASE em.SequenceStep OF
		
	1: 	TimerSim[1](PT := T#2S);
		TimerSim[1](in := TRUE);
		
		IF TimerSim[1].Q THEN
			em.Config.Data.I[1] := FALSE;
            em.Config.Data.I[2] := FALSE;
            em.Config.Data.I[3] := FALSE;
            em.Config.Data.I[4] := FALSE;
			TimerSim[1](in := FALSE);
		END_IF
		
	3: 	TimerSim[2](PT := T#2S);
		TimerSim[2](in := TRUE);
	
		IF TimerSim[2].Q THEN
			em.Config.Data.I[1] := TRUE;
			em.Config.Data.I[3] := TRUE;
			em.Config.Data.I[2] := FALSE;
			em.Config.Data.I[4] := FALSE;
			IF CmdSim THEN
				em.Cmd := E_CMD.reset;
			END_IF
			TimerSim[2](in := FALSE);
		END_IF
		
	4:	TimerSim[11](PT := T#1S);
		TimerSim[11](in := TRUE);
	
		IF TimerSim[11].Q THEN
			em.Config.Data.I[1] := TRUE;
			em.Config.Data.I[3] := TRUE;
			TimerSim[11](in := FALSE);
		END_IF
		
	5: 	TimerSim[3](PT := T#2S);
		TimerSim[3](in := TRUE);
		
		IF TimerSim[3].Q THEN
			em.Config.Data.I[1] := FALSE;
            em.Config.Data.I[2] := FALSE;
            em.Config.Data.I[3] := FALSE;
            em.Config.Data.I[4] := FALSE;
			TimerSim[3](in := FALSE);
		END_IF
	
	6:	IF CmdSim THEN
			TimerSim[4](PT := T#1S);
			TimerSim[4](in := TRUE);
		
			IF TimerSim[4].Q THEN
				em.Cmd := E_CMD.clear;
				TimerSim[4](in := FALSE);
			END_IF
		END_IF
		
	10: IF CmdSim THEN
			TimerSim[5](PT := T#1S);
			TimerSim[5](in := TRUE);
			IF TimerSim[5].Q THEN
				em.Cmd := E_CMD.start;
				TimerSim[5](in := FALSE);
			END_IF
		END_IF
	
	20:	TimerSim[6](PT := T#1S);
		TimerSim[6](in := TRUE);
		
		IF TimerSim[6].Q THEN
			IF CmdSim THEN
				em.Config.Data.I[5] := TRUE;
			END_IF
			TimerSim[6](in := FALSE);
		END_IF
		
	30: TimerSim[7](PT := T#2S);
		TimerSim[7](in := TRUE);
		
		IF TimerSim[7].Q THEN
			em.Config.Data.I[1] := FALSE;
			em.Config.Data.I[2] := TRUE;
			TimerSim[7](in := FALSE);
		END_IF
	
	40: TimerSim[8](PT := T#2S);
		TimerSim[8](in := TRUE);
		
		IF TimerSim[8].Q THEN
			em.Config.Data.I[3] := FALSE;
			em.Config.Data.I[4] := TRUE;
			TimerSim[8](in := FALSE);
		END_IF
		
	50:	TimerSim[12](PT := T#2S);
		TimerSim[12](in := TRUE);
		
		IF TimerSim[12].Q THEN
			em.Config.Data.I[4] := TRUE;
			TimerSim[12](in := FALSE);
		END_IF
		
	60:	TimerSim[9](PT := T#2S);
		TimerSim[9](in := TRUE);
		
		IF TimerSim[9].Q THEN
			IF CmdSim THEN
				em.Config.Data.I[5] := FALSE;
			END_IF
			TimerSim[9](in := FALSE);
		END_IF
	
	70: TimerSim[10](PT := T#2S);
		TimerSim[10](in := TRUE);
		
		IF TimerSim[10].Q THEN
			em.Config.Data.I[1] := TRUE;
			em.Config.Data.I[3] := TRUE;
			em.Config.Data.I[2] := FALSE;
			em.Config.Data.I[4] := FALSE;
			TimerSim[10](in := FALSE);
		END_IF
		
	
	END_CASE 
END_IF

END_FUNCTION_BLOCK

// ---- POUs/Sim/fbSignalSimPiotr.TcPOU
FUNCTION_BLOCK fbSignalSimPiotr
VAR_IN_OUT
	em : ARRAY[1..Counters.packmlEmLast] OF ST_EM;
	State : INT;
END_VAR
VAR_INPUT
	EnableSim : BOOL;
END_VAR
VAR
	timers : ARRAY[1..10] OF TON;
	sim : BOOL := TRUE;
END_VAR

IF EnableSim THEN
	CASE State OF
		40:	IF em[1].Config.Data.takeObject AND NOT em[1].Config.Data.objectSensor THEN
				em[1].Config.Data.objectSensor := TRUE;
			END_IF
			
		50:	IF em[2].Config.Data.takeObject AND NOT em[2].Config.Data.objectSensor THEN
				em[1].Config.Data.objectSensor := FALSE;
				em[2].Config.Data.objectSensor := TRUE;
			END_IF
			
		60:	IF em[3].Config.Data.takeObject AND NOT em[3].Config.Data.objectSensor THEN
				em[2].Config.Data.objectSensor := FALSE;
				em[3].Config.Data.objectSensor := TRUE;
			END_IF
			
		70:	IF em[4].Config.Data.takeObject AND NOT em[4].Config.Data.objectSensor THEN
				em[3].Config.Data.objectSensor := FALSE;
				em[4].Config.Data.objectSensor := TRUE;
			END_IF
			
		80:	IF em[2].Config.Data.takeObject AND NOT em[2].Config.Data.objectSensor THEN
				em[4].Config.Data.objectSensor := FALSE;
				em[2].Config.Data.objectSensor := TRUE;
			END_IF
			
		90:	IF em[5].Config.Data.takeObject AND NOT em[5].Config.Data.objectSensor THEN
				em[2].Config.Data.objectSensor := FALSE;
				em[5].Config.Data.objectSensor := TRUE;
			END_IF
			
		100:em[5].Config.Data.objectSensor := FALSE;
	END_CASE
END_IF

END_FUNCTION_BLOCK

// ---- DUTs/CM/Servo/fbCmServo.TcPOU
FUNCTION_BLOCK fbCmServo
VAR_IN_OUT
	em : ST_EM;
	cm : ST_CM_SERVO;
END_VAR
VAR
	
END_VAR

END_FUNCTION_BLOCK

// ---- POUs/UN/fbTaskPatrykUN.TcPOU
FUNCTION_BLOCK fbTaskPatrykUN EXTENDS fbUN
VAR	
	// Arrays with 'em' universal structure and 'fbEM' containing ST_MACHINE structure which contains of references to fbEM function block
	em : ARRAY[1..Counters.packmlEmLast] OF ST_EM;
	fbEM : ARRAY[1..Counters.packmlEmLast] OF ST_MACHINE;
	
	// Array containing all instances fo fbSliderEM with its own iterator
	SliderEM : ARRAY[1..Counters.SliderEMNo] OF fbSliderEM;
	iSliderEM : DINT := 1;
	
	// Array containing all instances fo fbSliderWithGripperEM with its own iterator
	SliderWithGripperEM : ARRAY[1..Counters.SliderWithGripperEMNo] OF fbSliderWithGripperEM;
	iSliderWithGripperEM : DINT := 1;
	
	// Array containing all instances fo fbXYMoverEM with its own iterator
	XYMoverEM : ARRAY[1..Counters.XYMoverEMNo] OF fbXYMoverEM;
	iXYMoverEM : DINT := 1;
	
	i : DINT;
	GlobalStep : INT := 0;
	NewStep : INT := 0;
	declareIterator : DINT;
	moduleWorkIterator : DINT;
	initIterator: DINT := 1;
	initialConfig: BOOL := TRUE;
	TimerOnSensor : TON;
	
	fbSignalSimXYMover : fbSignalSimXYMover;
	fbSignalSimSlider : fbSignalSimSlider;
	fbSignalSimSliderWithGripper : fbSignalSimSliderWithGripper;
	
END_VAR

//////////////////////////////////////////////////////////////////////
IF initialConfig THEN
	initialConfig := FALSE;
	
// Specifing module type of each module in array
em[1].Config.Functionality := E_Function.eSliderWithGripper;
em[2].Config.Functionality := E_Function.eSliderWithGripper;
em[3].Config.Functionality := E_Function.eSliderWithGripper;
em[4].Config.Functionality := E_Function.eSlider;
em[5].Config.Functionality := E_Function.eSlider;
em[6].Config.Functionality := E_Function.eSlider;
	
	// FOR loop to specify config for each module
FOR declareIterator := 1 TO Counters.packmlEmLast DO
	em[declareIterator].Config.Data.I REF= GVL.aInput[declareIterator];
	em[declareIterator].Config.Data.Q REF= GVL.aOutput[declareIterator];

	CASE em[declareIterator].Config.Functionality OF
		E_Function.eSlider:
			fbEM[declareIterator].fbEM REF= SliderEM[iSliderEM];
			iSliderEM := iSliderEM + 1;
		E_Function.eSliderWithGripper:
			fbEM[declareIterator].fbEM REF= SliderWithGripperEM[iSliderWithGripperEM];
			iSliderWithGripperEM := iSliderWithGripperEM + 1;
		E_Function.eXYMover:
			fbEM[declareIterator].fbEM REF= XYMoverEM[iXYMoverEM];
			iXYMoverEM := iXYMoverEM + 1;
	END_CASE
END_FOR
END_IF

FOR moduleWorkIterator := 1 TO Counters.packmlEmLast DO
	fbEM[moduleWorkIterator].fbEM(em := em[moduleWorkIterator], un := un, EnableSim := EnableSim, CmdSim := FALSE);
	
END_FOR

//////////////////////////////////////////////////////////////////////

IF cell.Cmd = E_CMD_CELL.STOP THEN
	GlobalStep := 100;
END_IF

IF cell.Cmd = E_CMD_CELL.ABORT THEN
	GlobalStep := 200;
END_IF

//////////////////////////////////////////////////////////////////////
//Deklaracja pick oraz drop pozycji
em[1].Config.Data.drop_pos := 2;
em[1].Config.Data.pick_pos := 1;
em[2].Config.Data.pick_pos := 3;
IF em[6].SequenceStep = 60 THEN
	em[2].Config.Data.drop_pos := 44;
	em[3].Config.Data.pick_pos := 54;
	ELSE
	em[2].Config.Data.drop_pos := 45;
	em[3].Config.Data.pick_pos := 55;	
END_IF
em[3].Config.Data.drop_pos := 6;

IF em[1].SequenceStep = 40 AND em[1].Config.Data.act_pos = 1 THEN
		TimerOnSensor(PT := T#1S);
		TimerOnSensor(IN := TRUE);
		IF TimerOnSensor.Q THEN
			em[1].Config.Data.I[3] := TRUE;
			TimerOnSensor(IN := FALSE);
		END_IF
END_IF

IF em[1].SequenceStep = 43 AND em[4].SequenceStep = 50 THEN
			em[1].Config.Data.I[3] := FALSE;
			em[4].Config.Data.I[3] := TRUE;
			GlobalStep := 32;
		END_IF

//////////////////////////////////////////////////////////////////////
CASE GlobalStep OF
	0:	un.Status := E_Status.undefined;
		GlobalStep := 10;
		
	10:	FOR i := 1 TO Counters.packmlEmLast DO
			IF NOT (em[i].Status = E_Status.idle) THEN
				un.Cmd := E_CMD.reset;
				RETURN;
			END_IF
		END_FOR
		un.Status := E_Status.idle;
		GlobalStep := 15;
		
	15:	IF cell.Cmd = E_CMD_CELL.START THEN
			un.Cmd := E_CMD.start;
			un.Status := E_Status.starting;
			GlobalStep := 20;
		END_IF
	
	20: FOR i := 1 TO Counters.packmlEmLast DO
			IF NOT (em[i].Status = E_Status.execute OR em[i].Status = E_Status.starting) THEN
				RETURN;
			END_IF
		END_FOR
		GlobalStep := 31;
	
	//30: IF em[1].SequenceStep = 40 AND em[4].SequenceStep = 50 THEN
			//em[1].Config.Data.I[3] := TRUE;
			//GlobalStep := 31;
		//END_IF
	
	31: IF em[1].SequenceStep = 43 AND em[4].SequenceStep = 50 THEN
			em[1].Config.Data.I[3] := FALSE;
			em[4].Config.Data.I[3] := TRUE;
			GlobalStep := 32;
		END_IF
		
	32: IF em[2].SequenceStep = 40 AND em[4].SequenceStep = 70 THEN
			em[4].Config.Data.I[3] := FALSE;
			GlobalStep := 40;
		END_IF
	
	40: IF em[2].Config.Data.drop_pos = 44 THEN
			GlobalStep := 51;
		ELSE
			GlobalStep := 41;
		END_IF
		
	41: IF em[2].SequenceStep = 40 AND em[3].SequenceStep = 40 THEN
			em[2].Config.Data.I[3] := TRUE;
			GlobalStep := 42;
		END_IF	
	
	42: IF em[2].SequenceStep = 43 THEN
			em[2].Config.Data.I[3] := FALSE;
			em[6].Config.Data.I[3] := TRUE;
			GlobalStep := 60;
		END_IF
		
	51: IF em[2].SequenceStep = 40 AND em[3].SequenceStep = 40 THEN
			em[2].Config.Data.I[3] := TRUE;
			GlobalStep := 52;
		END_IF
	
	52: IF em[2].SequenceStep = 43 THEN
			em[2].Config.Data.I[3] := FALSE;
			em[5].Config.Data.I[3] := TRUE;
			GlobalStep := 60;
		END_IF	
		
	60: IF em[6].SequenceStep = 70 THEN
			em[6].Config.Data.I[3] := FALSE;
			em[3].Config.Data.I[3] := TRUE;
			GlobalStep := 70;
		ELSIF em[5].SequenceStep = 70 THEN
			em[5].Config.Data.I[3] := FALSE;
			em[3].Config.Data.I[3] := TRUE;
			GlobalStep := 70;
		END_IF
		
	70:	IF em[3].SequenceStep = 43 THEN
			em[3].Config.Data.I[3] := FALSE;
			GlobalStep := 20;
		END_IF
	100: 	un.Cmd := E_Cmd.stop;
			un.Status := E_Status.stopping;
			GlobalStep := 101;		
	
	101: IF em[1].Status = E_Status.stopped AND em[2].Status = E_Status.stopped AND
			em[3].Status = E_Status.stopped AND em[4].Status = E_Status.stopped AND
			em[5].Status = E_Status.stopped AND em[6].Status = E_Status.stopped THEN
			un.Status := E_Status.stopped;
			GlobalStep := 10;
		END_IF
				
	200: un.Cmd := E_CMD.abort;
		 un.Status := E_Status.aborting;
		 GlobalStep := 201;
		
	201: IF em[1].Status = E_Status.aborted AND em[2].Status = E_Status.aborted AND
			em[3].Status = E_Status.aborted AND em[4].Status = E_Status.aborted AND
			em[5].Status = E_Status.aborted AND em[6].Status = E_Status.aborted THEN
			un.Status := E_Status.aborted;
			GlobalStep := 202;
		END_IF
		
		
	202: un.Cmd := E_CMD.clear;
		 GlobalStep := 10;
END_CASE

END_FUNCTION_BLOCK

// ---- GlobalTextList.TcGTLO
TEXTLIST GlobalTextList
  996 = '1'
  956 = '2'
  767 = '3'
  253 = '44'
  554 = '45'
  866 = '54'
  360 = '55'
  380 = '6'
  851 = 'Abort/Suspen'
  106 = 'Abort/Suspend'
  684 = 'Reset'
  686 = 'Start'
  366 = 'Stop/Hold'
END_TEXTLIST

// ---- VISUs/VisuPiotrUN.TcVIS
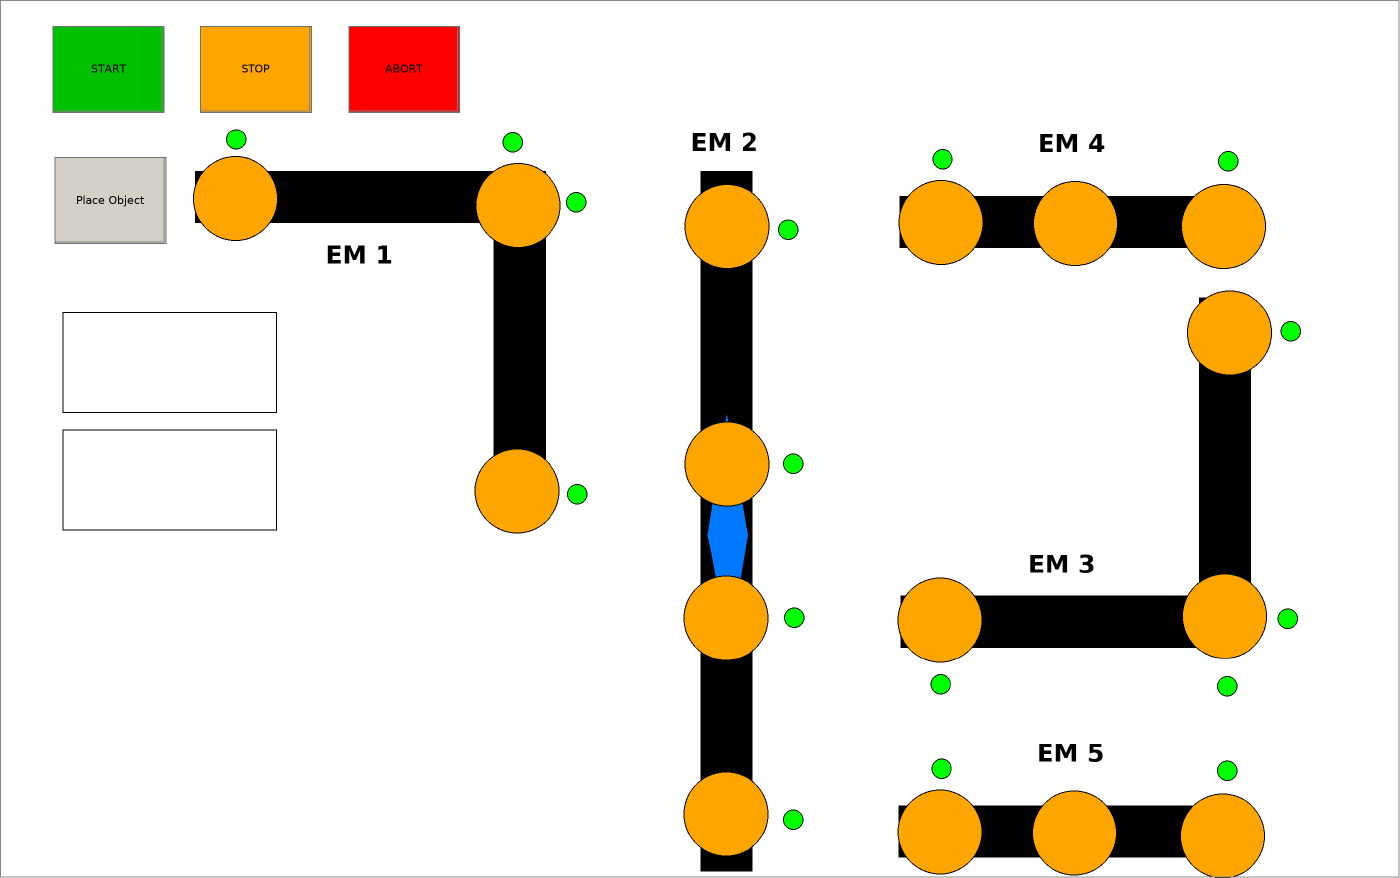
VISUALIZATION VisuPiotrUN  // 1407x883
    Rectangle (196,172 352x52)
    Rectangle (346,322 352x52), angle 90
    Button (55,158 112x87), "Place Object"
        toggle MAIN.cell.PlaceObject
    Ellipse (194,157 85x85), invisible if: NOT (MAIN.fbTaskPiotrUN.em[1].Config.Data.objectSensor AND MAIN.fbTaskPiotrUN.em[1].Config.Data.I[1])
    Button (53,26 112x87), "START"
        toggle MAIN.START
    Button (201,26 112x87), "STOP"
        toggle MAIN.STOP
    Button (350,26 112x87), "ABORT"
        toggle MAIN.ABORT
    Rectangle (378,498 704x52), angle 90
    Ellipse (688,185 85x85), invisible if: NOT (MAIN.fbTaskPiotrUN.em[2].Config.Data.I[3] AND MAIN.fbTaskPiotrUN.em[2].Config.Data.act_pos = 4)
    Ellipse (687,776 85x85), invisible if: NOT (MAIN.fbTaskPiotrUN.em[2].Config.Data.I[3] AND MAIN.fbTaskPiotrUN.em[2].Config.Data.act_pos = 1)
    Rectangle (1055,449 352x52), angle 90
    Rectangle (905,599 352x52)
    Rectangle (904,197 352x52)
    Ellipse (1187,185 85x85), invisible if: NOT (MAIN.fbTaskPiotrUN.em[4].StatusHMI.currentPositionWithObject = 1)
    Label (286,241 150x30), "EM 1"
    Label (653,128 150x30), "EM 2"
    Label (992,552 150x30), "EM 3"
    Polygon (711,538) (730,417) (751,538) (732,652) (716,562), invisible if: NOT (MAIN.fbTaskPiotrUN.em[2].Config.Data.act_pos = 666)
    Label (1002,129 150x30), "EM 4"
    Ellipse (688,424 85x85), invisible if: NOT (MAIN.fbTaskPiotrUN.em[2].Config.Data.I[3] AND MAIN.fbTaskPiotrUN.em[2].Config.Data.act_pos = 3)
    Ellipse (687,579 85x85), invisible if: NOT (MAIN.fbTaskPiotrUN.em[2].Config.Data.I[3] AND MAIN.fbTaskPiotrUN.em[2].Config.Data.act_pos = 2)
    Rectangle (63,432 215x101)
    Rectangle (63,314 215x101)
    Ellipse (505,133 20x20), invisible if: NOT MAIN.fbTaskPiotrUN.em[1].Config.Data.I[2]
    Ellipse (227,130 20x20), invisible if: NOT MAIN.fbTaskPiotrUN.em[1].Config.Data.I[1]
    Ellipse (570,487 20x20), invisible if: NOT MAIN.fbTaskPiotrUN.em[1].Config.Data.I[4]
    Ellipse (569,193 20x20), invisible if: NOT MAIN.fbTaskPiotrUN.em[1].Config.Data.I[3]
    Ellipse (937,150 20x20), invisible if: NOT (MAIN.fbTaskPiotrUN.em[4].StatusHMI.currentPosition = 2)
    Ellipse (1224,152 20x20), invisible if: NOT (MAIN.fbTaskPiotrUN.em[4].StatusHMI.currentPosition = 1)
    Ellipse (935,678 20x20), invisible if: NOT MAIN.fbTaskPiotrUN.em[3].Config.Data.I[1]
    Ellipse (1223,680 20x20), invisible if: NOT MAIN.fbTaskPiotrUN.em[3].Config.Data.I[2]
    Ellipse (1284,612 20x20), invisible if: NOT MAIN.fbTaskPiotrUN.em[3].Config.Data.I[3]
    Ellipse (1287,323 20x20), invisible if: NOT MAIN.fbTaskPiotrUN.em[3].Config.Data.I[4]
    Ellipse (782,221 20x20), invisible if: NOT (MAIN.fbTaskPiotrUN.em[2].Config.Data.act_pos = 4)
    Ellipse (787,456 20x20), invisible if: NOT (MAIN.fbTaskPiotrUN.em[2].Config.Data.act_pos = 3)
    Ellipse (788,611 20x20), invisible if: NOT (MAIN.fbTaskPiotrUN.em[2].Config.Data.act_pos = 2)
    Ellipse (787,814 20x20), invisible if: NOT ( MAIN.fbTaskPiotrUN.em[2].Config.Data.act_pos = 1)
    Ellipse (478,164 85x85), invisible if: NOT (MAIN.fbTaskPiotrUN.em[1].Config.Data.objectSensor AND MAIN.fbTaskPiotrUN.em[1].Config.Data.I[2] AND MAIN.fbTaskPiotrUN.em[1].Config.Data.I[3])
    Ellipse (477,451 85x85), invisible if: NOT (MAIN.fbTaskPiotrUN.em[1].Config.Data.objectSensor AND MAIN.fbTaskPiotrUN.em[1].Config.Data.I[4])
    Ellipse (1188,577 85x85), invisible if: NOT (MAIN.fbTaskPiotrUN.em[3].Config.Data.objectSensor AND MAIN.fbTaskPiotrUN.em[3].Config.Data.I[2] AND MAIN.fbTaskPiotrUN.em[3].Config.Data.I[3])
    Ellipse (902,581 85x85), invisible if: NOT (MAIN.fbTaskPiotrUN.em[3].Config.Data.objectSensor AND MAIN.fbTaskPiotrUN.em[3].Config.Data.I[1])
    Ellipse (1193,292 85x85), invisible if: NOT (MAIN.fbTaskPiotrUN.em[3].Config.Data.objectSensor AND MAIN.fbTaskPiotrUN.em[3].Config.Data.I[4])
    Ellipse (903,181 85x85), invisible if: NOT (MAIN.fbTaskPiotrUN.em[4].StatusHMI.currentPositionWithObject = 2)
    Ellipse (1038,182 85x85), invisible if: NOT MAIN.fbTaskPiotrUN.em[4].StatusHMI.isMovingWithObject
    Rectangle (903,810 352x52)
    Ellipse (1186,798 85x85), invisible if: NOT (MAIN.fbTaskPiotrUN.em[5].StatusHMI.currentPositionWithObject = 2)
    Label (1001,742 150x30), "EM 5"
    Ellipse (936,763 20x20), invisible if: NOT (MAIN.fbTaskPiotrUN.em[5].StatusHMI.currentPosition = 1)
    Ellipse (1223,765 20x20), invisible if: NOT (MAIN.fbTaskPiotrUN.em[5].StatusHMI.currentPosition = 2)
    Ellipse (902,794 85x85), invisible if: NOT (MAIN.fbTaskPiotrUN.em[5].StatusHMI.currentPositionWithObject = 1)
    Ellipse (1037,795 85x85), invisible if: NOT MAIN.fbTaskPiotrUN.em[5].StatusHMI.isMovingWithObject
END_VISUALIZATION
